SUBAPPLICATION VT_active (* Subapplication Type *)
  (* Standard: 61499-2 *)
  (* Version 1.0, 2023-02-19, franz *)
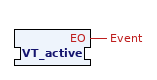
  EVENT_OUTPUT
    EO;
  END_EVENT
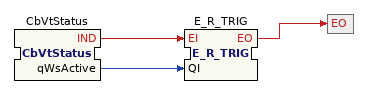
  FBS
    E_R_TRIG : E_R_TRIG;
    CbVtStatus : CbVtStatus;
  END_FBS
  EVENT_CONNECTIONS
    CbVtStatus.IND TO E_R_TRIG.EI;
    E_R_TRIG.EO TO EO;
  END_CONNECTIONS
  DATA_CONNECTIONS
    CbVtStatus.qWsActive TO E_R_TRIG.QI;
  END_CONNECTIONS
END_SUBAPPLICATION
